Fanuc KAREL source: kt00294.KL

PROGRAM KT00294
%STACKSIZE=65535
%PRIORITY=65535
%NOLOCKGROUP
VAR
I1 : INTEGER
R2 : REAL
OUT : BOOLEAN
BEGIN
I1=2
R2=3.0
-- UNSAFE_SOURCE_IR line 10: OUT = (R2 <> int_to_real(I1))
END KT00294
